FUNCTION_BLOCK FLASHER4
  (* Standard: 61499-2 *)
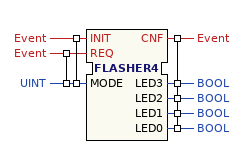
  EVENT_INPUT
    INIT WITH MODE;
    REQ WITH MODE;
  END_EVENT
  EVENT_OUTPUT
    CNF WITH LED3, LED2, LED1, LED0;
  END_EVENT
  VAR_INPUT
    MODE : UINT;
  END_VAR
  VAR_OUTPUT
    LED3 : BOOL;
    LED2 : BOOL;
    LED1 : BOOL;
    LED0 : BOOL;
  END_VAR
  VAR
    OFLO : BOOL;
  END_VAR
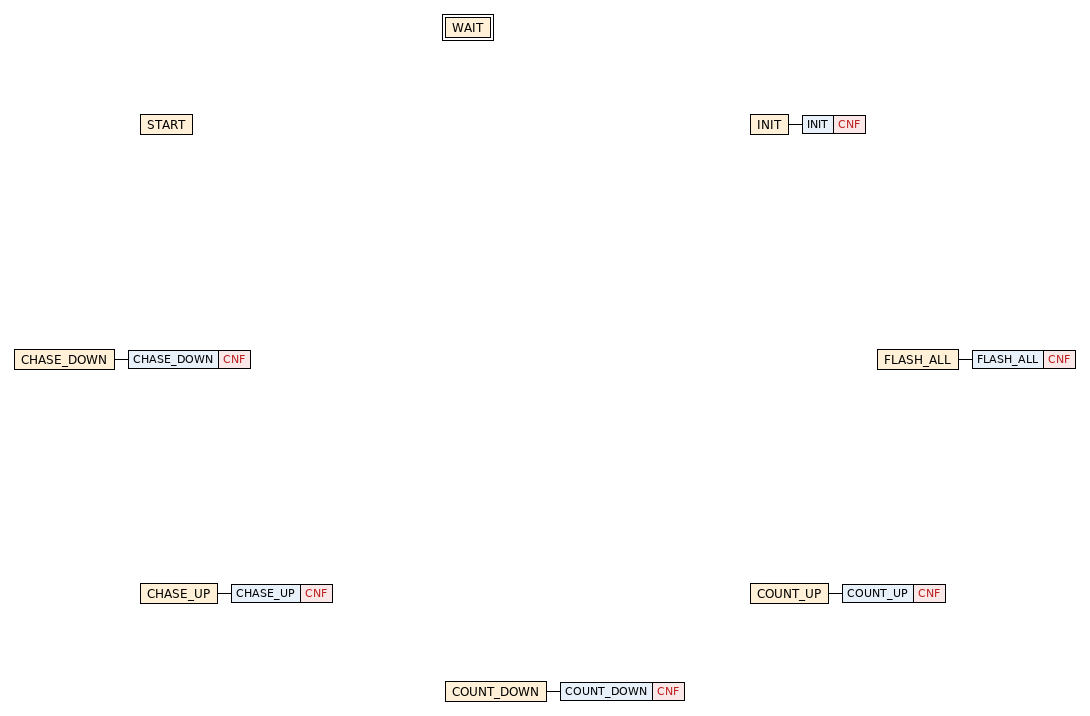
  EC_STATES
    WAIT;
    INIT : INIT -> CNF;
    FLASH_ALL : FLASH_ALL -> CNF;
    COUNT_UP : COUNT_UP -> CNF;
    COUNT_DOWN : COUNT_DOWN -> CNF;
    CHASE_UP : CHASE_UP -> CNF;
    CHASE_DOWN : CHASE_DOWN -> CNF;
    START;
  END_STATES
  EC_TRANSITIONS
    WAIT TO  := INIT;
    WAIT TO  := REQ;
    WAIT TO  := REQ;
    WAIT TO  := REQ;
    WAIT TO  := REQ;
    WAIT TO  := REQ;
    INIT TO  := 1;
    FLASH_ALL TO  := 1;
    COUNT_UP TO  := 1;
    COUNT_DOWN TO  := 1;
    CHASE_UP TO  := 1;
    CHASE_DOWN TO  := 1;
    START TO  := 1;
  END_TRANSITIONS
  ALGORITHM INIT IN ST:

  END_ALGORITHM
  ALGORITHM COUNT_UP IN ST:

  END_ALGORITHM
  ALGORITHM COUNT_DOWN IN ST:

  END_ALGORITHM
  ALGORITHM FLASH_ALL IN ST:

  END_ALGORITHM
  ALGORITHM CHASE_UP IN ST:

  END_ALGORITHM
  ALGORITHM CHASE_DOWN IN ST:

  END_ALGORITHM
END_FUNCTION_BLOCK
